FUNCTION_BLOCK FINAL FB_MiscOutput EXTENDS FB_EventLogger
VAR_INPUT
	Inhibit_Q				: BOOL;						//Inhibit Output
END_VAR                                             	
VAR_IN_OUT                                          	
	Control					: ST_System;            	//Machine Control Instance
END_VAR                                             	
VAR
	_Input		AT %I*		: BOOL;						//Raw Input 1
	_Auto					: BOOL;						//Auto of Output
	_ManOn					: BOOL;						//Manual On
	_ManOff					: BOOL;						//Manual Off
	_ForceOn				: BOOL;						//Force On
	_ForceOff				: BOOL;						//Force Off
	_Fault					: BOOL;						//Device Fault
	_OutputOn_ET			: REAL;						//Time output has been on since last being off
	_OutputOff_ET			: REAL;						//Time output has been off since last being on
	_FaultTimer_ET			: REAL;						//Fault timer elapsed
	_Alarm					: BOOL;						//Device Alarm
	_Warning				: BOOL;						//Device Warning
	_AlarmNum				: DINT;						//Device Alarm Number
	_WarningNum				: DINT;						//Device Warning Number
	_Value			AT %Q*	: BOOL;						//Value (physical output)                                         	
	_R_Trig					: ARRAY[0..9] OF R_TRIG;	//Private Rising Edge Triggers
END_VAR
VAR PERSISTENT
	_Name					: STRING[15];				//Name for HMI
	_Description			: STRING[40];				//Description for HMI
	_AlarmMute				: BOOL;						//Alarm Mute
	_CycleCount				: DINT;						//Total cycles
	_FaultTimer_PT			: REAL;						//Fault timer preset time
END_VAR

M_AlarmMonitor();
M_WarningMonitor();
M_UnlatchManuals();
M_SetOutput();

//Calculate time output has been on/off since last change
IF _Value THEN
	_OutputOn_ET := _OutputOn_ET + Control.SystemTime.ScanTime;
	_OutputOff_ET := 0;
ELSE
	_OutputOff_ET := _OutputOff_ET + Control.SystemTime.ScanTime;
	_OutputOn_ET := 0;
END_IF;

{attribute 'monitoring' := 'variable'}
PROPERTY PUBLIC Alarm : Bool
GET
Alarm := _Alarm;
END_GET
END_PROPERTY

{attribute 'monitoring' := 'variable'}
PROPERTY PUBLIC AlarmMute : BOOL
SET
AlarmMute := _AlarmMute;
END_SET
END_PROPERTY

{attribute 'monitoring' := 'variable'}
PROPERTY PUBLIC Auto : Bool
GET // PUBLIC
Auto := _Auto;
END_GET
SET
_Auto := Auto;
END_SET
END_PROPERTY

{attribute 'monitoring' := 'variable'}
PROPERTY PUBLIC CycleCount : DINT
GET
CycleCount := _CycleCount;
END_GET
END_PROPERTY

{attribute 'monitoring' := 'variable'}
PROPERTY PUBLIC Description : String[40]
GET
Description := _Description;
END_GET
SET
_Description := Description;
END_SET
END_PROPERTY

{attribute 'monitoring' := 'variable'}
PROPERTY PUBLIC Fault : Bool
SET
_Fault := Fault;
END_SET
END_PROPERTY

{attribute 'monitoring' := 'variable'}
PROPERTY PUBLIC FaultTimer_ET : real
GET
FaultTimer_ET := _FaultTimer_ET;
END_GET
END_PROPERTY

{attribute 'monitoring' := 'variable'}
PROPERTY PUBLIC FaultTimer_PT : real
GET
FaultTimer_PT := _FaultTimer_PT;
END_GET
SET
_FaultTimer_PT := FaultTimer_PT;
END_SET
END_PROPERTY

{attribute 'monitoring' := 'variable'}
PROPERTY PUBLIC ForceOff : Bool
GET
ForceOff := _ForceOff;
END_GET
SET
_ForceOff := ForceOff;
END_SET
END_PROPERTY

{attribute 'monitoring' := 'variable'}
PROPERTY PUBLIC ForceOn : Bool
GET
ForceOn := _ForceOn;
END_GET
SET
_ForceOn := ForceOn;
END_SET
END_PROPERTY

{attribute 'monitoring' := 'variable'}
PROPERTY PUBLIC Input : Bool
GET
Input := _Input;
END_GET
END_PROPERTY

METHOD PRIVATE M_AlarmMonitor
VAR_INPUT
END_VAR
VAR_INST
END_VAR
VAR_INST // added by the converter: edge detectors and wires of the graphical bodies
    _w1, _w2, _w3 : BOOL;
    _rt1 : R_TRIG;
END_VAR
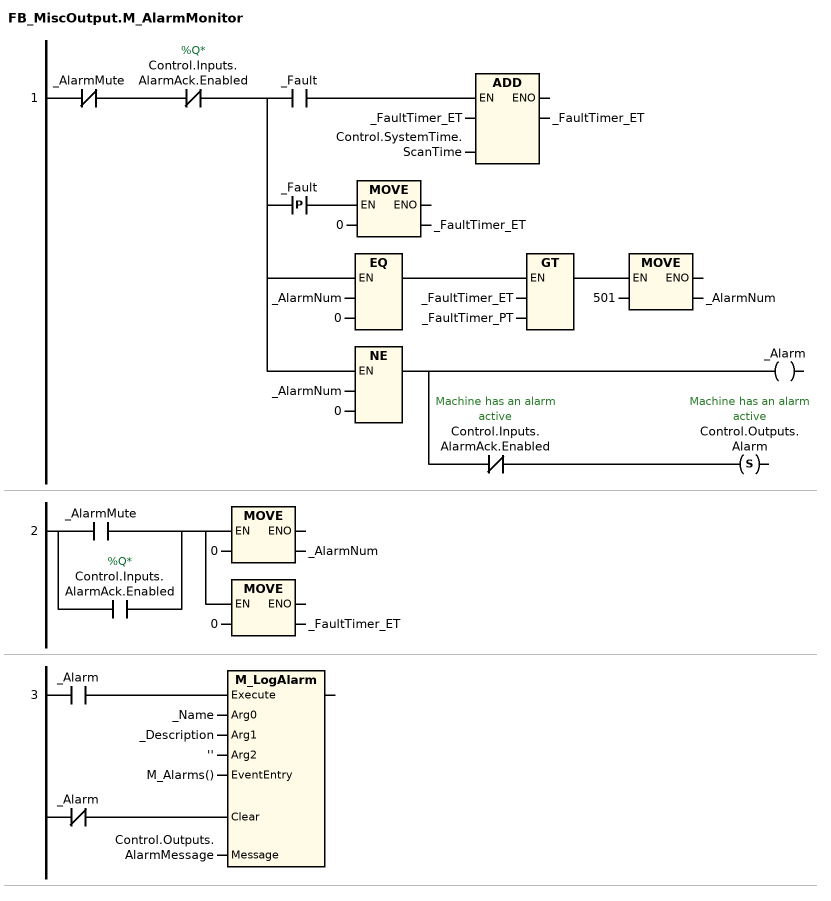
// NETWORK 1
//   Control.Inputs.AlarmAck.Enabled: AT %Q* | Machine has an alarm active
//   _FaultTimer_ET: Fault timer elapsed
//   Control.SystemTime.ScanTime: Last scan time (Seconds)
//   _FaultTimer_PT: Fault timer preset time
//   Control.Outputs.Alarm: Machine has an alarm active
_w1 := NOT _AlarmMute AND NOT Control.Inputs.AlarmAck.Enabled;
IF _w1 AND _Fault THEN _FaultTimer_ET := _FaultTimer_ET + Control.SystemTime.ScanTime; END_IF
_rt1(CLK := _Fault);
IF _w1 AND _rt1.Q THEN _FaultTimer_ET := 0; END_IF
IF _w1 AND _AlarmNum = 0 AND _FaultTimer_ET > _FaultTimer_PT THEN _AlarmNum := 501; END_IF
_w2 := _w1 AND _AlarmNum <> 0;
_Alarm := _w2;
Control.Outputs.Alarm S= _w2 AND NOT Control.Inputs.AlarmAck.Enabled;

// NETWORK 2
//   Control.Inputs.AlarmAck.Enabled: AT %Q*
//   _FaultTimer_ET: Fault timer elapsed
_w3 := _AlarmMute OR Control.Inputs.AlarmAck.Enabled;
IF _w3 THEN _AlarmNum := 0; END_IF
IF _w3 THEN _FaultTimer_ET := 0; END_IF

// NETWORK 3
M_LogAlarm(Execute := _Alarm, Arg0 := _Name, Arg1 := _Description, Arg2 := '', EventEntry := M_Alarms(), Clear := NOT _Alarm, Message := Control.Outputs.AlarmMessage);
END_METHOD

METHOD PRIVATE M_Alarms : TcEventEntry
VAR_INPUT
END_VAR
CASE _AlarmNum OF
	501: M_Alarms:= TC_Events.TcMiscOutput.A_501;//Alarm				
ELSE
	M_Alarms:= TC_Events.TcMiscOutput.A_Undefined;
END_CASE
END_METHOD

METHOD PRIVATE M_SetOutput
VAR
END_VAR
VAR_INST
END_VAR
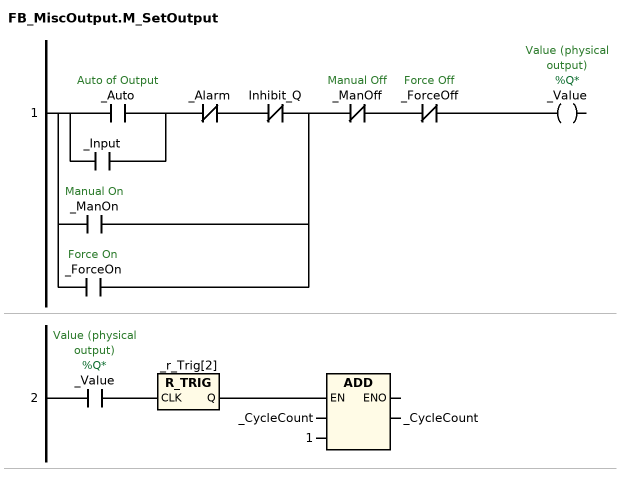
// NETWORK 1
//   _Auto: Auto of Output
//   _ManOn: Manual On
//   _ForceOn: Force On
//   _ManOff: Manual Off
//   _ForceOff: Force Off
//   _Value: Value (physical output) | AT %Q*
_Value := ((_Auto OR _Input) AND NOT _Alarm AND NOT Inhibit_Q OR _ManOn OR _ForceOn) AND NOT _ManOff AND NOT _ForceOff;

// NETWORK 2
//   _Value: Value (physical output) | AT %Q*
//   _CycleCount: Total cycles
_r_Trig[2](CLK := _Value); // R_TRIG
IF _r_Trig[2].Q THEN _CycleCount := _CycleCount + 1; END_IF
END_METHOD

METHOD PRIVATE M_UnlatchManuals
VAR_INPUT
END_VAR
VAR_INST
END_VAR
VAR_INST // added by the converter: edge detectors and wires of the graphical bodies
    _rt1, _rt2, _rt3 : R_TRIG;
END_VAR
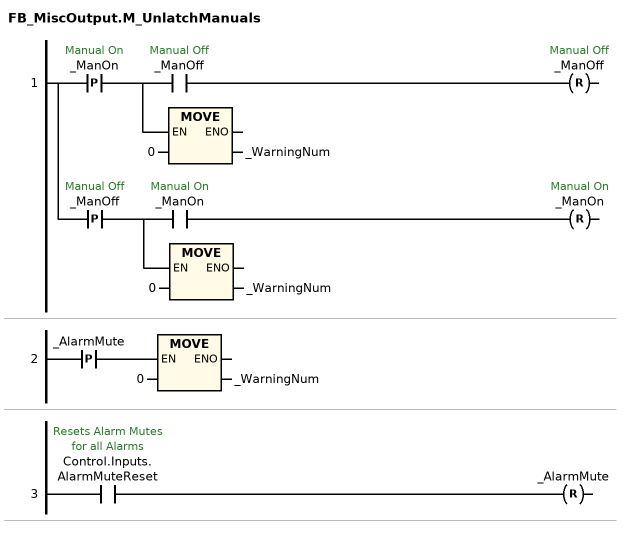
// NETWORK 1
//   _ManOn: Manual On
//   _ManOff: Manual Off
_rt1(CLK := _ManOn);
_ManOff R= _rt1.Q AND _ManOff;
IF _rt1.Q THEN _WarningNum := 0; END_IF
_rt2(CLK := _ManOff);
_ManOn R= _rt2.Q AND _ManOn;
IF _rt2.Q THEN _WarningNum := 0; END_IF

// NETWORK 2
_rt3(CLK := _AlarmMute);
IF _rt3.Q THEN _WarningNum := 0; END_IF

// NETWORK 3
//   Control.Inputs.AlarmMuteReset: Resets Alarm Mutes for all Alarms
_AlarmMute R= Control.Inputs.AlarmMuteReset;
END_METHOD

METHOD PRIVATE M_WarningMonitor
VAR_INPUT
END_VAR
VAR_INST
END_VAR
VAR_INST // added by the converter: edge detectors and wires of the graphical bodies
    _w1, _w2 : BOOL;
END_VAR
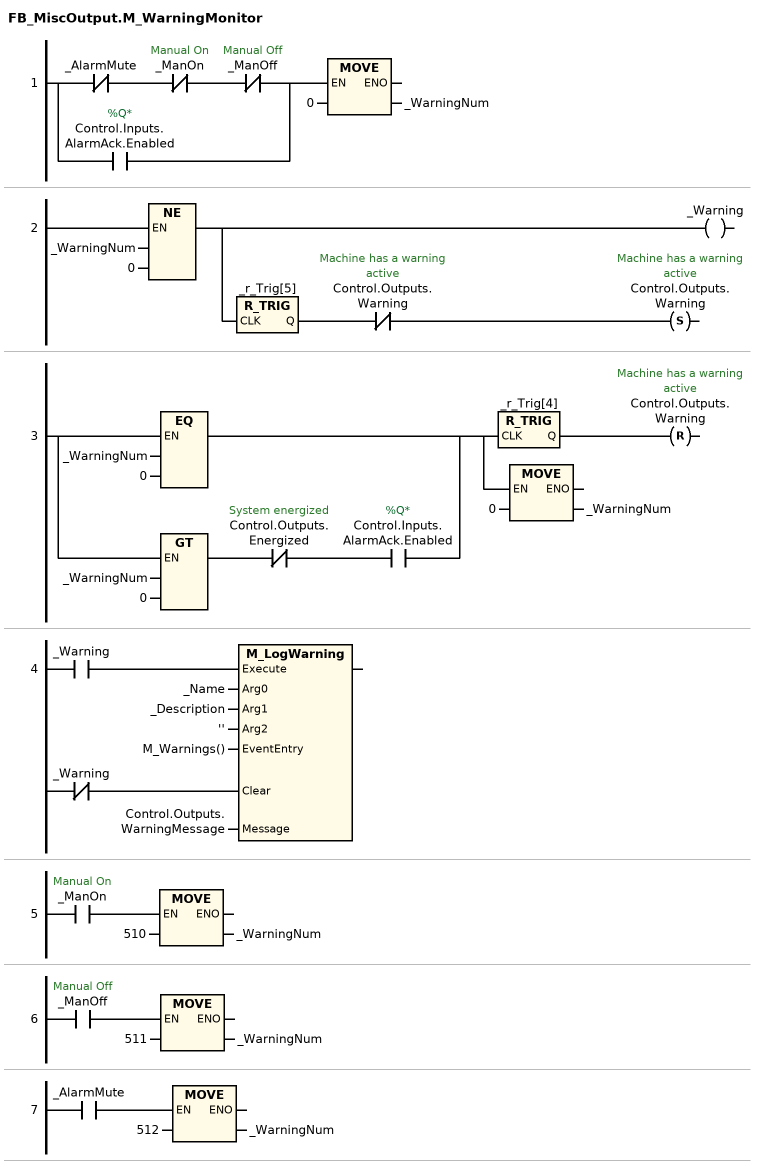
// NETWORK 1
//   _ManOn: Manual On
//   _ManOff: Manual Off
//   Control.Inputs.AlarmAck.Enabled: AT %Q*
IF NOT _AlarmMute AND NOT _ManOn AND NOT _ManOff OR Control.Inputs.AlarmAck.Enabled THEN _WarningNum := 0; END_IF

// NETWORK 2
//   Control.Outputs.Warning: Machine has a warning active
_w1 := _WarningNum <> 0;
_Warning := _w1;
_r_Trig[5](CLK := _w1); // R_TRIG
Control.Outputs.Warning S= _r_Trig[5].Q AND NOT Control.Outputs.Warning;

// NETWORK 3
//   Control.Outputs.Energized: System energized
//   Control.Inputs.AlarmAck.Enabled: AT %Q*
//   Control.Outputs.Warning: Machine has a warning active
_w2 := _WarningNum = 0 OR _WarningNum > 0 AND NOT Control.Outputs.Energized AND Control.Inputs.AlarmAck.Enabled;
_r_Trig[4](CLK := _w2); // R_TRIG
Control.Outputs.Warning R= _r_Trig[4].Q;
IF _w2 THEN _WarningNum := 0; END_IF

// NETWORK 4
M_LogWarning(Execute := _Warning, Arg0 := _Name, Arg1 := _Description, Arg2 := '', EventEntry := M_Warnings(), Clear := NOT _Warning, Message := Control.Outputs.WarningMessage);

// NETWORK 5
//   _ManOn: Manual On
IF _ManOn THEN _WarningNum := 510; END_IF

// NETWORK 6
//   _ManOff: Manual Off
IF _ManOff THEN _WarningNum := 511; END_IF

// NETWORK 7
IF _AlarmMute THEN _WarningNum := 512; END_IF
END_METHOD

METHOD PRIVATE M_Warnings : TcEventEntry
VAR_INPUT
END_VAR
CASE _WarningNum OF
	510: M_Warnings:= TC_Events.TcMiscOutput.W_510;//Manual ON
	511: M_Warnings:= TC_Events.TcMiscOutput.W_511;//Manual OFF		
	512: M_Warnings:= TC_Events.TcMiscOutput.W_512;//Alarm Mute Active						
ELSE
	M_Warnings:=  TC_Events.TcMiscOutput.W_Undefined;
END_CASE
END_METHOD

{attribute 'monitoring' := 'variable'}
PROPERTY PUBLIC ManOff : Bool
GET
ManOff := _ManOff;
END_GET
SET
_ManOff := ManOff;
END_SET
END_PROPERTY

{attribute 'monitoring' := 'variable'}
PROPERTY PUBLIC ManOn : Bool
GET
ManOn := _ManOn;
END_GET
SET
_ManOn := ManOn;
END_SET
END_PROPERTY

{attribute 'monitoring' := 'variable'}
PROPERTY PUBLIC Name : String[15]
GET
Name := _Name;
END_GET
SET
_Name := Name;
END_SET
END_PROPERTY

{attribute 'monitoring' := 'variable'}
PROPERTY PUBLIC OutputOff_ET : real
GET
OutputOff_ET := _OutputOff_ET;
END_GET
END_PROPERTY

{attribute 'monitoring' := 'variable'}
PROPERTY PUBLIC OutputOn_ET : real
GET
OutputOn_ET := _OutputOn_ET;
END_GET
END_PROPERTY

{attribute 'monitoring' := 'variable'}
PROPERTY PUBLIC StandbyReset : Bool
GET
StandbyReset := _ForceOff;
END_GET
SET
_ForceOff := StandbyReset;
END_SET
END_PROPERTY

{attribute 'monitoring' := 'variable'}
PROPERTY PUBLIC Value : Bool
GET
Value := _Value;
END_GET
SET
_Value := Value;
END_SET
END_PROPERTY

{attribute 'monitoring' := 'variable'}
PROPERTY PUBLIC Warning : Bool
GET
Warning := _Warning;
END_GET
END_PROPERTY

END_FUNCTION_BLOCK

(* stored: Version 1.1.0.1, ProductVersion 3.1.4024.3
   POU FB_MiscOutput: Id {1b94a963-190f-497b-94ed-5541ca9049ca}, SpecialFunc None
   Property Alarm: Id {a477ff6b-08f7-4ee8-968d-fd970896a9e5}
   Get Get: Id {007875d2-9d25-4544-a7fb-f7ae52ee60d7}
   Property AlarmMute: Id {713ad340-eb86-4ce3-9893-aaa9c3a975dc}
   Set Set: Id {07d662c0-2162-4d64-88a6-f819d7e728cc}
   Property Auto: Id {8116078f-6d41-474b-8d6e-806aace94bfa}
   Get Get: Id {cd0140d0-f417-4c1a-b1f9-4e135acdab2a}
   Set Set: Id {744a6dc9-981e-442d-b153-cb4bf98db8e0}
   Property CycleCount: Id {ed706daf-deab-4d25-9094-91f2fc81081b}
   Get Get: Id {fda000e8-3a51-4abc-931b-dd57dfe82092}
   Property Description: Id {325e421f-2052-455e-aab1-3b4d93eb1965}
   Get Get: Id {9e393bc2-7f11-4aa6-ae95-a25843e05787}
   Set Set: Id {c1bfd63f-30bc-4e0e-95d9-f2a1ab7725ca}
   Property Fault: Id {9a59b6f7-3c1f-4275-b798-7836844580f4}
   Set Set: Id {ac9c41f9-6e75-4381-9b16-2dde70556329}
   Property FaultTimer_ET: Id {1d58687a-52d9-4717-b20a-8e1d6ea7862d}
   Get Get: Id {23c447fb-4682-48cc-a663-f358db1bb8fd}
   Property FaultTimer_PT: Id {91d355c0-5979-4759-9ac9-8b206a30a5ee}
   Get Get: Id {6c659ad2-04a8-4b35-90ca-e48f5cbcbaa6}
   Set Set: Id {12ea5cb0-a475-439d-9c94-20b0089e3946}
   Property ForceOff: Id {3498bff8-7282-4b24-b73f-18fd1c1c2dc4}
   Get Get: Id {7e3b4ce5-b18a-488c-8126-54532f2957bd}
   Set Set: Id {43685ff4-b708-4e40-9fe8-f40b2fd813c9}
   Property ForceOn: Id {f5075e5c-5b13-491a-94fd-053f59c44619}
   Get Get: Id {0a622389-0361-4186-9484-4ed48460cc27}
   Set Set: Id {82433792-8986-4308-b48a-c83696b0cb84}
   Property Input: Id {856476ef-a4be-4130-958a-f61a6f0f65aa}
   Get Get: Id {a8831c48-eb24-42a8-9a88-afa7569acf41}
   Method M_AlarmMonitor: Id {0d6d681c-4788-4b5b-b945-56506c62a4bd}
   Method M_Alarms: Id {bee028b9-2dd7-4e23-bf89-45010f7482a8}
   Method M_SetOutput: Id {2e3c5ed2-0df2-4349-8890-eb5f4c6c5367}
   Method M_UnlatchManuals: Id {4e54a148-40a7-487f-81df-dfc0e1629bf8}
   Method M_WarningMonitor: Id {22c7063f-c53e-4630-9c16-3f2fcceca4fb}
   Method M_Warnings: Id {19d6d8bd-c268-4a42-95a4-7f698e702d98}
   Property ManOff: Id {7b83616d-053e-4ab3-84b1-27dca58e9ee7}
   Get Get: Id {b39c0b49-5c90-40c0-a444-1e90e6853a53}
   Set Set: Id {8fd10089-3b09-4789-a75a-06c686fcded8}
   Property ManOn: Id {374ecd19-f50a-448a-9a34-4416eb172dad}
   Get Get: Id {915e4c9c-c844-4a72-8e9b-137b95260184}
   Set Set: Id {2a7f26ca-a42d-4e31-8d1d-d3af48866025}
   Property Name: Id {05911eca-2c71-4b9d-9e28-1f1783f8d564}
   Get Get: Id {37fb887e-0223-4125-ac26-4df6483efa32}
   Set Set: Id {75096810-2ee8-47ac-a182-5505881779d1}
   Property OutputOff_ET: Id {43164add-c0ab-4db6-99f2-2de018e0e939}
   Get Get: Id {a46231b6-fff4-4ddf-8a2e-df5df60b9ce1}
   Property OutputOn_ET: Id {35df065b-6956-428a-b1e2-d18b1d033872}
   Get Get: Id {c3ca6aa9-a0ef-4d5b-af60-b275e7097137}
   Property StandbyReset: Id {c3e305f5-d7e8-4cbd-bd9f-96ed2a49c636}
   Get Get: Id {4e71149d-9ae6-4e09-a1df-6679331095d0}
   Set Set: Id {f945f155-a38c-4b16-a945-d4b5689c8361}
   Property Value: Id {d0d70c14-2f3f-45cc-a1c2-e77f5b11d8df}
   Get Get: Id {ba4c2828-e005-44bc-aaa3-17b43fbeeb74}
   Set Set: Id {82e29c90-0e31-472e-bb78-9a0c18158e8c}
   Property Warning: Id {4f574a59-0a0b-4c7b-8de9-8af8f8c75d7b}
   Get Get: Id {8667b6b4-1e0e-415c-a14f-25ad1635ccfc} *)
